FUNCTION_BLOCK FB_MotionAxisDS402 IMPLEMENTS I_MotionAxis
VAR_INPUT
END_VAR
VAR_OUTPUT
END_VAR
VAR
        AxisRef : REFERENCE TO AXIS_REF;
        bRestoreDone : BOOL;
        bRestoreError : BOOL;
        bRestoreErrorID : UDINT;
END_VAR

IF NOT __ISVALIDREF( AxisRef ) THEN
    RETURN;
END_IF

{warning 'Add property implementation'}
PROPERTY AxisState : MC_AxisStates
GET
END_GET
SET
END_SET
END_PROPERTY

{warning 'Add property implementation'}
PROPERTY Busy : BOOL
GET
END_GET
SET
END_SET
END_PROPERTY

{warning 'Add method implementation '}
METHOD CalibrateEncValue
END_METHOD

{warning 'Add property implementation'}
PROPERTY Cmd : UINT
GET
END_GET
SET
END_SET
END_PROPERTY

{warning 'Add property implementation'}
PROPERTY CmdData : UINT
GET
END_GET
SET
END_SET
END_PROPERTY

{warning 'Add method implementation '}
METHOD CyclicCalls
END_METHOD

{warning 'Add property implementation'}
PROPERTY Done : BOOL
GET
END_GET
SET
END_SET
END_PROPERTY

METHOD EncErrorCheck : BOOL
VAR_INPUT
    EncError : BOOL;
    EncErrorCode : UDINT;
END_VAR
END_METHOD

{warning 'Add method implementation '}
METHOD EncSaveRestore
END_METHOD

{warning 'Add property implementation'}
PROPERTY Error : BOOL
GET
END_GET
SET
END_SET
END_PROPERTY

{warning 'Add property implementation'}
PROPERTY ErrorCode : BOOL
GET
END_GET
SET
END_SET
END_PROPERTY

{warning 'Add method implementation '}
METHOD ErrorHandling
END_METHOD

//FB_Init is always available implicitly and it is used primarily for initialization.
//The return value is not evaluated. For a specific influence, you can also declare the
//methods explicitly and provide additional code there with the standard initialization
//code. You can evaluate the return value.
METHOD FB_Init: BOOL
VAR_INPUT
    bInitRetains: BOOL; // TRUE: the retain variables are initialized (reset warm / reset cold)
    bInCopyCode: BOOL;  // TRUE: the instance will be copied to the copy code afterward (online change)
    AxisReference : REFERENCE TO AXIS_REF;
END_VAR
AxisRef REF= AxisReference;
END_METHOD

{warning 'Add method implementation '}
METHOD GearIn
END_METHOD

{warning 'Add method implementation '}
METHOD GearOut
END_METHOD

{warning 'Add method implementation '}
METHOD GetAxisRef : REFERENCE TO AXIS_REF
END_METHOD

{warning 'Add method implementation '}
METHOD GetPowerOverride : LREAL
END_METHOD

{warning 'Add method implementation '}
METHOD Halt
VAR_INPUT
    Deceleration	: LREAL := 0.0;
    Jerk	: LREAL := 0.0;
    BufferMode	: MC_BufferMode := .MC_BufferMode.MC_Aborting;
END_VAR
VAR_OUTPUT
    Done	: BOOL;
    Busy	: BOOL;
    Active	: BOOL;
    CommandAborted	: BOOL;
    Error	: BOOL;
    ErrorID	: UDINT;
    ErrorStr	: T_MaxString;
END_VAR
END_METHOD

{warning 'Add property implementation'}
PROPERTY HaltBusy : BOOL
GET
END_GET
END_PROPERTY

{warning 'Add property implementation'}
PROPERTY HaltDone : BOOL
GET
END_GET
END_PROPERTY

{warning 'Add property implementation'}
PROPERTY HaltError : BOOL
GET
END_GET
END_PROPERTY

{warning 'Add property implementation'}
PROPERTY HaltErrorID : UDINT
GET
END_GET
END_PROPERTY

{warning 'Add method implementation '}
METHOD Home
END_METHOD

{warning 'Add property implementation'}
PROPERTY HomeBusy : BOOL
GET
END_GET
SET
END_SET
END_PROPERTY

{warning 'Add property implementation'}
PROPERTY HomeDone : BOOL
GET
END_GET
SET
END_SET
END_PROPERTY

{warning 'Add property implementation'}
PROPERTY HomeError : BOOL
GET
END_GET
SET
END_SET
END_PROPERTY

{warning 'Add property implementation'}
PROPERTY HomeErrorID : UDINT
GET
END_GET
SET
END_SET
END_PROPERTY

{warning 'Add property implementation'}
PROPERTY HomeMode : E_EpicsHomeCmd
GET
END_GET
SET
END_SET
END_PROPERTY

{warning 'Add property implementation'}
PROPERTY HomePosition : LREAL
GET
END_GET
SET
END_SET
END_PROPERTY

{warning 'Add property implementation'}
PROPERTY MeasuredAcceleration : LREAL
GET
END_GET
END_PROPERTY

{warning 'Add property implementation'}
PROPERTY MeasuredPosition : LREAL
GET
END_GET
END_PROPERTY

{warning 'Add property implementation'}
PROPERTY MeasuredVelocity : LREAL
GET
END_GET
END_PROPERTY

{warning 'Add method implementation '}
METHOD MoveAbsolute
VAR_INPUT
    Position	: LREAL;
    Velocity	: LREAL;
    Acceleration	: LREAL := 0.0;
    Deceleration	: LREAL := 0.0;
    Jerk	: LREAL := 0.0;
    BufferMode	: MC_BufferMode := .MC_BufferMode.MC_Aborting;
END_VAR
VAR_OUTPUT
    Done	: BOOL;
    Busy	: BOOL;
    Active	: BOOL;
    CommandAborted	: BOOL;
    Error	: BOOL;
    ErrorID	: UDINT;
    ErrorStr	: T_MaxString;
END_VAR
END_METHOD

{warning 'Add property implementation'}
PROPERTY MoveAbsoluteBusy : BOOL
GET
END_GET
END_PROPERTY

{warning 'Add property implementation'}
PROPERTY MoveAbsoluteDone : BOOL
GET
END_GET
END_PROPERTY

{warning 'Add property implementation'}
PROPERTY MoveAbsoluteError : BOOL
GET
END_GET
END_PROPERTY

{warning 'Add property implementation'}
PROPERTY MoveAbsoluteErrorID : UDINT
GET
END_GET
END_PROPERTY

{warning 'Add property implementation'}
PROPERTY MoveAbsoluteTargetAcceleration : LREAL
GET
END_GET
END_PROPERTY

{warning 'Add property implementation'}
PROPERTY MoveAbsoluteTargetDeceleration : LREAL
GET
END_GET
END_PROPERTY

{warning 'Add property implementation'}
PROPERTY MoveAbsoluteTargetJerk : LREAL
GET
END_GET
END_PROPERTY

{warning 'Add property implementation'}
PROPERTY MoveAbsoluteTargetPosition : LREAL
GET
END_GET
END_PROPERTY

{warning 'Add property implementation'}
PROPERTY MoveAbsoluteTargetVelocity : LREAL
GET
END_GET
END_PROPERTY

{warning 'Add property implementation'}
PROPERTY Name : STRING
GET
END_GET
SET
END_SET
END_PROPERTY

{warning 'Add property implementation'}
PROPERTY NegativeMotionIsEnabled : BOOL
GET
END_GET
END_PROPERTY

{warning 'Add property implementation'}
PROPERTY Override : LREAL
GET
END_GET
SET
END_SET
END_PROPERTY

{warning 'Add property implementation'}
PROPERTY PositiveMotionIsEnabled : BOOL
GET
END_GET
END_PROPERTY

{warning 'Add method implementation '}
METHOD Power
VAR_INPUT
    Enable	: BOOL;
    Enable_Positive	: BOOL;
    Enable_Negative	: BOOL;
    (* in percent from 0 to 100 *)
    Override	: LREAL := 100.0;
    BufferMode	: MC_BufferMode := .MC_BufferMode.MC_Aborting;
END_VAR
VAR_OUTPUT
    Status	: BOOL;
    Busy	: BOOL;
    Active	: BOOL;
    Error	: BOOL;
    ErrorID	: UDINT;
    ErrorStr	: T_MaxString;
END_VAR
END_METHOD

{warning 'Add property implementation'}
PROPERTY PowerError : BOOL
GET
END_GET
END_PROPERTY

{warning 'Add property implementation'}
PROPERTY PowerErrorID : UDINT
GET
END_GET
END_PROPERTY

{warning 'Add property implementation'}
PROPERTY PowerIsEnabled : BOOL
GET
END_GET
END_PROPERTY

{warning 'Add property implementation'}
PROPERTY PowerOverride : LREAL
GET
END_GET
END_PROPERTY

{warning 'Add property implementation'}
PROPERTY PowerSelf : BOOL
GET
END_GET
SET
END_SET
END_PROPERTY

{warning 'Add property implementation'}
PROPERTY PowerStatus : BOOL
GET
END_GET
END_PROPERTY

{warning 'Add method implementation '}
METHOD Resetting
VAR_OUTPUT
    Done	: BOOL;
    Busy	: BOOL;
    Error	: BOOL;
    ErrorID	: UDINT;
    ErrorStr	: T_MaxString;
END_VAR
END_METHOD

{warning 'Add property implementation'}
PROPERTY RestoreDone : BOOL
GET
END_GET
SET
END_SET
END_PROPERTY

{warning 'Add property implementation'}
PROPERTY RestoreError : BOOL
GET
END_GET
SET
END_SET
END_PROPERTY

{warning 'Add property implementation'}
PROPERTY RestoreErrorID : UDINT
GET
END_GET
SET
END_SET
END_PROPERTY

{warning 'Add property implementation'}
PROPERTY SetpointAcceleration : LREAL
GET
END_GET
END_PROPERTY

{warning 'Add property implementation'}
PROPERTY SetpointJerk : LREAL
GET
END_GET
END_PROPERTY

{warning 'Add property implementation'}
PROPERTY SetpointPosition : LREAL
GET
END_GET
END_PROPERTY

{warning 'Add property implementation'}
PROPERTY SetpointVelocity : LREAL
GET
END_GET
END_PROPERTY

{warning 'Add method implementation '}
METHOD SetPowerOverride
VAR_INPUT
    (* in percent from 0 to 100 *)
    Override	: LREAL;
END_VAR
VAR_OUTPUT
    Status	: BOOL;
    Busy	: BOOL;
    Active	: BOOL;
    Error	: BOOL;
    ErrorID	: UDINT;
    ErrorStr	: T_MaxString;
END_VAR
END_METHOD

METHOD SetRestorePosition : BOOL
VAR_INPUT
    Load : BOOL;
    Position : LREAL;
END_VAR
END_METHOD

{warning 'Add property implementation'}
PROPERTY TargetReached : BOOL
GET
END_GET
SET
END_SET
END_PROPERTY

END_FUNCTION_BLOCK

(* stored: Version 1.1.0.1
   POU FB_MotionAxisDS402: Id {e6939303-1a29-4526-8cba-ad7b7e0a797c}, SpecialFunc None
   Property AxisState: Id {f2c10954-6fbf-47cd-a4c6-2595e49dff9a}
   Get Get: Id {21390da1-2c90-444d-8ca2-bcc7f982732a}
   Set Set: Id {21a42741-3163-48b4-85ca-487a70b81ddc}
   Property Busy: Id {be5040ac-8ff2-4ec4-93df-83ebd8969c60}
   Get Get: Id {7ed734b0-29b8-442a-975e-fc096e88aa06}
   Set Set: Id {26aac89d-deb6-4042-8ca7-a740c6a46515}
   Method CalibrateEncValue: Id {c7dcbcfa-a780-4c13-83ee-dd3a3259e8a3}
   Property Cmd: Id {1b379d54-0a62-44d6-a8e8-4d08c001a496}
   Get Get: Id {0498f7e8-8844-4c9e-90cd-6b596e76e1d3}
   Set Set: Id {b9abc620-d0f5-4548-8d50-0eefc66b482c}
   Property CmdData: Id {fd172632-bf45-4562-936c-a14063505d37}
   Get Get: Id {d55567f2-f174-4f99-b639-de4ce227069a}
   Set Set: Id {82e2542e-c0c9-41e9-ac90-ee42aae6dc01}
   Method CyclicCalls: Id {5caaab68-ed2c-4395-b4aa-32b1b31e9573}
   Property Done: Id {51fa4c87-afdd-47a9-8ad1-66b50ff00d39}
   Get Get: Id {48eb093d-9bb9-4989-a9a6-52ae56edd306}
   Set Set: Id {000710c8-060d-48d1-9a80-6fafe0682e03}
   Method EncErrorCheck: Id {750c3ad0-4f69-4f01-ad1d-777d71f8e0df}
   Method EncSaveRestore: Id {758fc86b-abf1-47a5-8f0f-d4ef3c0ab63d}
   Property Error: Id {cac518e7-c4c8-4f02-a58c-d3e7d2d79cd8}
   Get Get: Id {1f4a15a1-4924-401f-9889-63882261a5e7}
   Set Set: Id {47d8c067-a717-4f6d-a286-220187089055}
   Property ErrorCode: Id {0921f86d-40cd-4df8-ab28-2898c44fa05e}
   Get Get: Id {8966b06b-b307-481c-b0a4-39b5860997da}
   Set Set: Id {3b89c017-0708-43e9-a767-4c8bb2b97e00}
   Method ErrorHandling: Id {bccf0ad9-f658-4128-bd0e-a1c0b1f3a9b5}
   Method FB_Init: Id {180fa942-a7f1-463e-8d13-f7f31c42583f}
   Method GearIn: Id {bd71ffe0-808b-46c3-b7c4-4726451849e9}
   Method GearOut: Id {2f2fbcf8-48b9-4907-94c3-c4b4bd82d7a2}
   Method GetAxisRef: Id {70970299-6294-431d-9776-54d7232b96ee}
   Method GetPowerOverride: Id {49fbbd23-2407-4a66-ae5b-2e18cb4981be}
   Method Halt: Id {0d0d9db3-d251-4c98-9ee5-9c7cabbfae92}
   Property HaltBusy: Id {d5f36f64-1a55-4d41-a9c2-c76317220329}
   Get Get: Id {42083908-85a4-4f3d-92af-233c0686bc20}
   Property HaltDone: Id {d9c4a5e0-2ab3-40f5-9994-0eb6f9d01433}
   Get Get: Id {d16c9e22-5d30-483a-b808-c9aae656db15}
   Property HaltError: Id {5cfd0afa-c6b4-4b7b-b1d8-bb124ec37fdc}
   Get Get: Id {25e8bafc-b207-40a1-a2ef-9cefff41729c}
   Property HaltErrorID: Id {786f40cf-1067-458f-98f2-6541393330db}
   Get Get: Id {3b06a852-b6f5-475c-9fc8-4862cb335a53}
   Method Home: Id {c1e21c0a-478a-4e64-ac1c-4da91135d244}
   Property HomeBusy: Id {0b614afd-f884-405d-a3c9-940069cf0094}
   Get Get: Id {223b0e5f-eb6e-47c2-a3c7-5787f373de75}
   Set Set: Id {7be8f0f9-f51a-454d-a887-5d28f4efed94}
   Property HomeDone: Id {71a6249c-03b6-4d17-9f52-bb3ed3787205}
   Get Get: Id {ad2908a1-2ddd-4a33-9355-57e43968bd13}
   Set Set: Id {a12dad95-1663-46f2-89bc-5b943fb0f647}
   Property HomeError: Id {7bff45de-d38d-4489-8fcf-0f584a5ea1d2}
   Get Get: Id {08b2d4a1-b885-4442-9e3f-55fa2ad595c0}
   Set Set: Id {70843d1c-fd3b-4247-a647-d87861efc7d2}
   Property HomeErrorID: Id {96ec42bb-ae64-4aa5-9cd2-f55a53d0dc8d}
   Get Get: Id {4406e833-cc87-4d1f-9954-9da0df4b5de6}
   Set Set: Id {45471b98-d625-420f-849b-16bb662bd4e7}
   Property HomeMode: Id {3abfb9b6-6330-4090-937f-149b0df774d9}
   Get Get: Id {51b06faf-ec66-4c42-bfcd-78f3784b0816}
   Set Set: Id {a45435ca-380e-47b0-afc7-bff58a7a751b}
   Property HomePosition: Id {e14099f4-0519-4f8c-bebc-835ed61738a8}
   Get Get: Id {79fd6318-2139-4df7-95ce-4f71625ca4ba}
   Set Set: Id {eeecc061-37e6-4eda-b549-072f5d48d7d0}
   Property MeasuredAcceleration: Id {934d9697-a40f-4eb9-a7f7-67ee6985cc2f}
   Get Get: Id {e0ab7cc1-6634-4353-9667-b1c724ec3f2d}
   Property MeasuredPosition: Id {2a84fca6-0f9b-4280-b2ca-2049fcfb94bd}
   Get Get: Id {a6a4bb59-026a-4928-9c9b-df4598680652}
   Property MeasuredVelocity: Id {efb2b425-b568-4bdf-833b-5bc65db366a5}
   Get Get: Id {cda91a7e-e3af-4435-9ed1-45de112df9a3}
   Method MoveAbsolute: Id {b79a8962-0b6c-4e26-8a83-40993f407295}
   Property MoveAbsoluteBusy: Id {0790109c-56c3-4e19-b6c2-acb92c392cb4}
   Get Get: Id {3d201901-9a75-4553-a5fa-ff6fe54d4d7a}
   Property MoveAbsoluteDone: Id {faeaacd2-8a9d-415c-9a78-e670be07b3d2}
   Get Get: Id {7f54dfdf-b07b-43f6-a310-d8d65b8720b6}
   Property MoveAbsoluteError: Id {4e493c61-094a-4389-995a-30e3946962cd}
   Get Get: Id {ed3b3d18-5d2e-4637-86ea-b9254eb9d0c5}
   Property MoveAbsoluteErrorID: Id {17e71446-17ad-4326-9132-290dafd4cf95}
   Get Get: Id {5ef70246-ab88-49b6-9f00-b8346a776b02}
   Property MoveAbsoluteTargetAcceleration: Id {642747c5-2103-4fe7-a4be-f191a1d64a90}
   Get Get: Id {cc1dfd9e-5ea9-416b-ab11-d1f7798db597}
   Property MoveAbsoluteTargetDeceleration: Id {e3db52ec-2501-41b8-b3ec-7be41fd21e1b}
   Get Get: Id {5eda09d2-41e2-4a9e-90b3-b7124ee9a43a}
   Property MoveAbsoluteTargetJerk: Id {70798a58-70dc-4808-a405-d9ca44e190c1}
   Get Get: Id {686b5815-904d-4225-bc40-f7da9e53721d}
   Property MoveAbsoluteTargetPosition: Id {2c8be390-cc7e-4683-9c6c-e00b2832638d}
   Get Get: Id {634b2890-d916-4ecb-be59-0a3fd804b486}
   Property MoveAbsoluteTargetVelocity: Id {9aff5306-41b3-4638-9345-15453e87a59d}
   Get Get: Id {0f80d99b-6f11-4c05-a4ea-dea851e710c2}
   Property Name: Id {c639e75a-3678-46d3-9835-47292b8528fe}
   Get Get: Id {fbaabfdf-504e-49ca-8875-601d5bac9ee2}
   Set Set: Id {7f3715a1-94d8-4ff9-ba44-9f5b8814b5c9}
   Property NegativeMotionIsEnabled: Id {7436ed1f-8644-4767-a7b5-08e16f5bc0a0}
   Get Get: Id {82bdc18b-2a7d-4d47-9621-01a7daccf2f2}
   Property Override: Id {7ea85e17-c860-400c-8c06-481a9966edfc}
   Get Get: Id {b56989ed-8e9d-41f5-98d5-be9d080a592a}
   Set Set: Id {4fc3e807-232c-4e8c-97b0-34cf39465a4e}
   Property PositiveMotionIsEnabled: Id {138ca617-0311-48a2-b19f-9e05794a76aa}
   Get Get: Id {f8bacf70-521b-46ae-879e-223de80f5c38}
   Method Power: Id {19d5d4aa-b380-44c1-a057-53da5a253fbc}
   Property PowerError: Id {68e594af-d141-444e-90dd-82d59426c017}
   Get Get: Id {13ad7120-04ca-4246-8e27-b7d429f86465}
   Property PowerErrorID: Id {e51792b2-d6f8-4544-a4f6-a19a4ee87bed}
   Get Get: Id {7bf2a67f-e3f8-4a07-bc29-e7f263650237}
   Property PowerIsEnabled: Id {2378d27c-639d-4a59-acb6-f7785b054605}
   Get Get: Id {1c39cdf1-d58d-47fd-8958-e56759420fbf}
   Property PowerOverride: Id {276994d9-1b30-4079-a978-8003304548f3}
   Get Get: Id {899ce412-1fd3-4721-8996-5169d30d1796}
   Property PowerSelf: Id {9d14efce-1b7d-49a8-8025-76afc49ffec8}
   Get Get: Id {37b34cfb-5d2b-4009-84a8-398befd21f8f}
   Set Set: Id {7781505d-ef97-4cd1-bcdf-dd756d369879}
   Property PowerStatus: Id {7a605967-f92b-43b5-8bb0-9eb4ff790479}
   Get Get: Id {fb0c8156-d81b-4a08-982e-f83282b7374a}
   Method Resetting: Id {3a445482-f12e-4a74-b8f7-8f9d0d15c6fe}
   Property RestoreDone: Id {cb765afb-1413-4429-925c-810a8dd64bb7}
   Get Get: Id {84627456-aefe-4341-a2e2-ecb57c435076}
   Set Set: Id {edb638d1-76d7-42a9-8dc8-51939e63d9cd}
   Property RestoreError: Id {ce78b1c5-487b-4bf4-822d-fe41f5c45005}
   Get Get: Id {50fdf11a-e66d-4772-86ae-e3ebc54d547a}
   Set Set: Id {05a703b3-1fa1-4f7f-896a-f5105867dc22}
   Property RestoreErrorID: Id {138430a3-2ab5-40ed-b4d6-ca237265df5c}
   Get Get: Id {d3b74895-4801-4acb-bda9-5ecfb0946553}
   Set Set: Id {58c1ef80-9e86-47a6-ae2b-217ed7c48851}
   Property SetpointAcceleration: Id {2b173762-6328-4e4c-95a8-b0b12612577c}
   Get Get: Id {d5868310-b848-4212-9134-fbd16e577603}
   Property SetpointJerk: Id {cb34f141-25c4-4329-957c-2f43fad59182}
   Get Get: Id {d9db7ea2-f8ce-4019-8c3c-40fdaa823278}
   Property SetpointPosition: Id {646f602a-22b9-4e57-88d7-81645cf1ef98}
   Get Get: Id {c7b5ce4f-fd1c-4607-8ae3-2f7f9a9d315c}
   Property SetpointVelocity: Id {75af3429-3580-4fd1-aa71-20f5f83b23b6}
   Get Get: Id {f94d94cf-9d1a-440b-a311-94bd32652378}
   Method SetPowerOverride: Id {d2b8fabe-aac6-4f1a-a530-9a80a3f12907}
   Method SetRestorePosition: Id {7727cf9a-f768-466b-9368-d638fbcdb1f7}
   Property TargetReached: Id {fc4e962e-2148-4171-88f4-52555729e5f9}
   Get Get: Id {1fe3d58e-990f-42c5-8d94-e39c038d5344}
   Set Set: Id {5bc7028a-0343-4c6f-aff2-3fd174ee4f61} *)
